// TIA Portal V19 export
FUNCTION_BLOCK "MwFakCalc_FB"   // FB145, LAD
TITLE = COIL CAR
// stored: MemoryReserve 100, SetENOAutomatically false
   VAR_INPUT
      AreaInterface : "AreaInterface";
      ZSI : "udt_ZoneSafetyInterface";
      DSI : Struct
         PushAx : "udt_DeviceSafetyInterface";
         Gripper : "udt_DeviceSafetyInterface";
      END_STRUCT;
      Drive : Struct
         PushAx : "TAx_DriveInterface";
      END_STRUCT;
      HWID : Struct
         PushAx_TEL1 : HW_SUBMODULE;
      END_STRUCT;
      DataIn : Struct
         MaterialPresenceEntry : Bool;
         MaterialPresenceExit : Bool;
         MaterialJam : Bool;
         PushAx_Ls_HomeFwd : Bool;
         PushAx_Ls_RestBwd : Bool;
         PushAx_Ls_LowSpeedHome : Bool;
         PushAx_Ls_LowSpeedRest : Bool;
         PushAx_Ls_Touch : Bool;
         Gripper_Ls_ForceOpen : Bool;   // TRUE = Movable supprts must be closed
         PushAx : "SpeedMachine_DataIn";
         Gripper : "ValveMachine_DataIn";
      END_STRUCT;
      CIn : Struct
         Manager : Struct
            EnableStopDoorOpeningReq : Bool;
            EnableStopInPhase : Bool;
            EnableStopProgrammed : Bool;
         END_STRUCT;
         Rollformer_Standstill : Bool;
         Rollformer_CheckNextFwd : Bool;
         Rollformer_CheckNextBwd : Bool;
         MW_ActualFAK : LReal;
         SemiAut_And_ButtonPressed : Bool;
         PostServo_MeasuredValueG : LReal;
         PostServo_MeasuredValueW : LReal;
         PostServo_MeasuredID : UInt;
      END_STRUCT;
      Config : Struct
         PushAx : "SpeedMachine_Config";
         Gripper : "ValveMachine_Config";
         MaterialPresenceDly : Time;
         MaterialAbsenceDly : Time;
         PushAx_FwdTimeout { ExternalAccessible := 'False'; ExternalVisible := 'False'; ExternalWritable := 'False'} : Time;
         PushAx_BwdTimeout { ExternalAccessible := 'False'; ExternalVisible := 'False'; ExternalWritable := 'False'} : Time;
         Default_FAK : LReal;
      END_STRUCT;
   END_VAR
   VAR_OUTPUT
      MachineInterface : "MachineInterface";
      DataOut : Struct
         PushAx : "SpeedMachine_DataOut";
         Gripper : "ValveMachine_DataOut";
         MeasInput_ExeReg : Bool;
      END_STRUCT;
      COut : Struct
         PushAx : "SpeedMachine_COut";
         Gripper : "ValveMachine_COut";
         StopMaterialFeeding : Bool;
         MW_FAK_ChangeIsRequest : Bool;
      END_STRUCT;
   END_VAR
   VAR_IN_OUT
      PersistentValues : "udt_MwFacCalc_Pers";
      TO_Gripper_Encoder : TO_ExternalEncoder;
      TO_Gripper_MeasInput : TO_MeasuringInput;
      TO_Wheel_MeasInput : TO_MeasuringInput;
   END_VAR
   VAR
      Sts : Struct
         PushAx : Struct
            LowSpeedRest : Bool;
            LowSpeedHome : Bool;
         END_STRUCT;
         Gripper : Struct
            OffsetPos : LReal;
            PosRel : LReal;
         END_STRUCT;
         AlarmPresence : Bool;
         Status : Int;
         MW_FAK_ChangeIsRequest : Bool;
         AverageFAKIsValid : Bool;
         WheelMeasInp_SaveIdLastPosEdge : UInt;
         GripperMeasInp_SaveIdLastPosEdge : UInt;
         GripperMeasInp_LastID : UInt;
         WheelMeasInp_LastID : UInt;
         PostServo_LastID : UInt;
      END_STRUCT;
      Ctrl : Struct
         StopInPhase : Bool;
         StopProgrammed : Bool;
         MeasuringStart : Bool;
         MeasInp_Enable : Bool;
         Meas1_Exe : Bool;
         Meas2_Exe : Bool;
         Gripper_RollformerForceOpen : Bool;
         Gripper_AutOpen : Bool;
         Gripper_AutClose : Bool;
         PushAx_AutFwd : Bool;
         PushAx_AutBwd : Bool;
         Rollformer_FwdEnable : Bool;
         Rollformer_BkwWnable : Bool;
         Rollformer_FastStop : Bool;
      END_STRUCT;
      Alarm : Struct
         PushAx_UnvalidStateLsZeroRest : Bool;
         PushAx_UnvalidStateLsLow : Bool;
         PushAx_LowSpeedHome_NotEngaged : Bool;
         PushAx_LowSpeedRest_NotEngaged : Bool;
         PushAx_TimeoutFwd : Bool;
         PushAx_TimeoutBwd : Bool;
         MaterialNoPresence : Bool;
         MaterialJamEntry : Bool;
         Meas1RegNotGet : Bool;
         Meas2RegNotGet : Bool;
         Gripper_MaxPosExceed : Bool;
         PushAx : "SpeedMachine_Alr";
         Gripper : "ValveAlr";
         Gripper_Encoder : "TExtEncoder_Alarms";
         Gripper_MeasInput : "TMeasuring_Alarms";
         Wheel_MeasInput : "TMeasuring_Alarms";
      END_STRUCT;
      Warning : Struct
         PushAx : "SpeedMachine_Wng";
         Gripper : "ValveMachine_Wng";
         MaterialNoPrresence : Bool;
      END_STRUCT;
      Diag : Struct
         Gripper_Encoder : "TO_Diagnostic";
         Gripper_MeasInput : "TO_Diagnostic";
         Wheel_MeasInput : "TO_Diagnostic";
      END_STRUCT;
      PushAx : "SpeedMachine_FB";
      Gripper : "ValveMachine_FB";
      Gripper_MeasInp { S7_SetPoint := 'True'} : "MeasuringInput";
      Wheel_MeasInp { S7_SetPoint := 'True'} : "MeasuringInput";
      MeasRegIEmpty { S7_SetPoint := 'True'} : "udt_MwFacCalc_RegItem";
      tonMaterialPresence : TON_TIME;
      tonMaterialAbsence : TON_TIME;
      tonPushAxFwd { S7_SetPoint := 'True'} : TON_TIME;
      tonPushAxBwd { S7_SetPoint := 'True'} : TON_TIME;
      tonRollformer_BwdCheckNext { S7_SetPoint := 'True'} : TON_TIME;
   END_VAR
   VAR_TEMP
      i : Int;
      Delta_W : LReal;
      Delta_G : LReal;
      FAK_Acc : LReal;
      Tol : LReal;
      LongerPartLength_ActualFAK : LReal;
      LongerPartLength_NewFAK : LReal;
   END_VAR
BEGIN

REGION Network 1 (SCL): Reset alarms command

   IF #AreaInterface.RstAlarms THEN
       // Alarms
       #Alarm.PushAx_UnvalidStateLsZeroRest := FALSE;
       #Alarm.PushAx_UnvalidStateLsLow := FALSE;
       #Alarm.PushAx_LowSpeedHome_NotEngaged := FALSE;
       #Alarm.PushAx_LowSpeedRest_NotEngaged := FALSE;
       #Alarm.PushAx_TimeoutFwd := FALSE;
       #Alarm.PushAx_TimeoutBwd := FALSE;
       #Alarm.MaterialNoPresence := FALSE;
       #Alarm.MaterialJamEntry := FALSE;
       #Alarm.Meas1RegNotGet := FALSE;
       #Alarm.Meas2RegNotGet := FALSE;
       #Alarm.Gripper_MaxPosExceed := FALSE;

   END_IF;
END_REGION

REGION Network 3: Material Presence
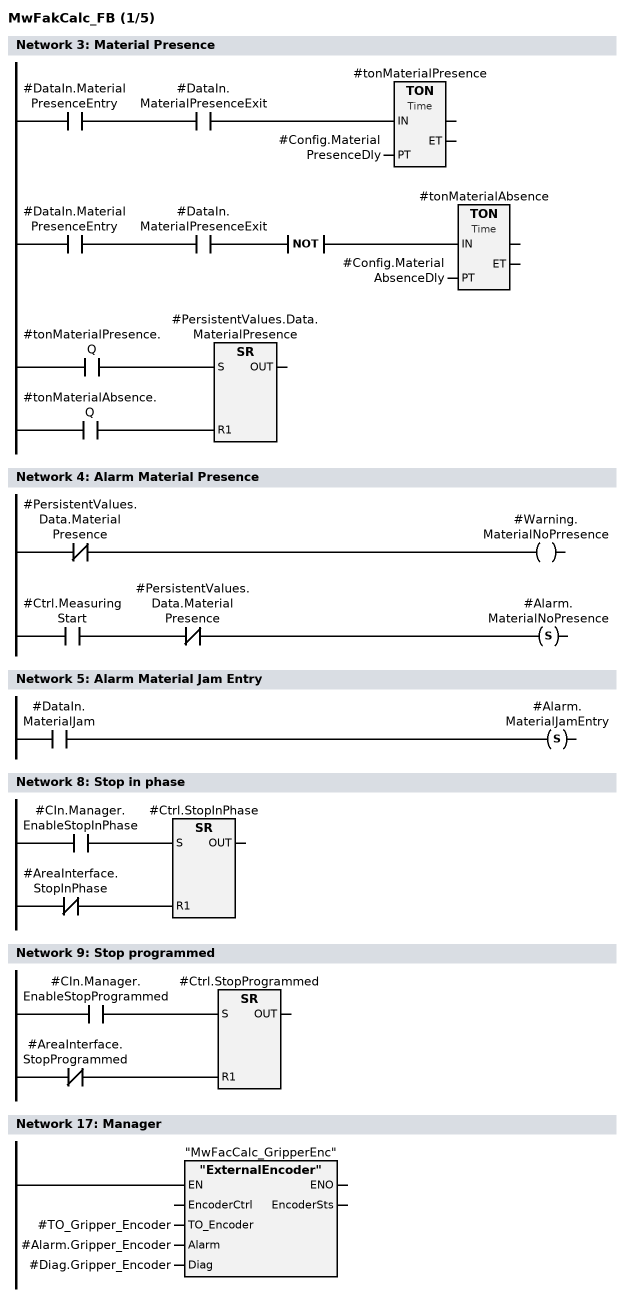
   RUNG wire#powerrail
      Contact( #DataIn.MaterialPresenceEntry )
      Contact( #DataIn.MaterialPresenceExit )
      { S7_Templates := "time_type := Time" } #tonMaterialPresence.TON(pt := #Config.MaterialPresenceDly, et =>)
   END_RUNG
   RUNG wire#powerrail
      Contact( #DataIn.MaterialPresenceEntry )
      Contact( #DataIn.MaterialPresenceExit )
      Not()
      { S7_Templates := "time_type := Time" } #tonMaterialAbsence.TON(pt := #Config.MaterialAbsenceDly, et =>)
   END_RUNG
   RUNG wire#powerrail
      Contact( #tonMaterialPresence.Q )
      S_SR(operand := #PersistentValues.Data.MaterialPresence, r1 := wire#w1)
   END_RUNG
   RUNG wire#powerrail
      Contact( #tonMaterialAbsence.Q )
   END_RUNG wire#w1
   // the same network as SCL:
   #tonMaterialPresence(IN := #DataIn.MaterialPresenceEntry AND #DataIn.MaterialPresenceExit,   // TON
                        PT := #Config.MaterialPresenceDly);
   #tonMaterialAbsence(IN := NOT (#DataIn.MaterialPresenceEntry AND #DataIn.MaterialPresenceExit),   // TON
                       PT := #Config.MaterialAbsenceDly);
   IF #tonMaterialPresence.Q THEN
       #PersistentValues.Data.MaterialPresence := TRUE;   // SR flip-flop
   END_IF;
   IF #tonMaterialAbsence.Q THEN #PersistentValues.Data.MaterialPresence := FALSE; END_IF;
END_REGION

REGION Network 4: Alarm Material Presence
   RUNG wire#powerrail
      I_Contact( #PersistentValues.Data.MaterialPresence )
      Coil( #Warning.MaterialNoPrresence )
   END_RUNG
   RUNG wire#powerrail
      Contact( #Ctrl.MeasuringStart )
      I_Contact( #PersistentValues.Data.MaterialPresence )
      S_Coil( #Alarm.MaterialNoPresence )
   END_RUNG
   // the same network as SCL:
   #Warning.MaterialNoPrresence := NOT #PersistentValues.Data.MaterialPresence;
   IF #Ctrl.MeasuringStart AND NOT #PersistentValues.Data.MaterialPresence THEN
       #Alarm.MaterialNoPresence := TRUE;
   END_IF;
END_REGION

REGION Network 5: Alarm Material Jam Entry
   RUNG wire#powerrail
      Contact( #DataIn.MaterialJam )
      S_Coil( #Alarm.MaterialJamEntry )
   END_RUNG
   // the same network as SCL:
   IF #DataIn.MaterialJam THEN #Alarm.MaterialJamEntry := TRUE; END_IF;
END_REGION

REGION Network 7: <<<CYCLE >>>
END_REGION

REGION Network 8: Stop in phase
   RUNG wire#powerrail
      Contact( #CIn.Manager.EnableStopInPhase )
      S_SR(operand := #Ctrl.StopInPhase, r1 := wire#w1)
   END_RUNG
   RUNG wire#powerrail
      I_Contact( #AreaInterface.StopInPhase )
   END_RUNG wire#w1
   // the same network as SCL:
   IF #CIn.Manager.EnableStopInPhase THEN
       #Ctrl.StopInPhase := TRUE;   // SR flip-flop
   END_IF;
   IF NOT #AreaInterface.StopInPhase THEN #Ctrl.StopInPhase := FALSE; END_IF;
END_REGION

REGION Network 9: Stop programmed
   RUNG wire#powerrail
      Contact( #CIn.Manager.EnableStopProgrammed )
      S_SR(operand := #Ctrl.StopProgrammed, r1 := wire#w1)
   END_RUNG
   RUNG wire#powerrail
      I_Contact( #AreaInterface.StopProgrammed )
   END_RUNG wire#w1
   // the same network as SCL:
   IF #CIn.Manager.EnableStopProgrammed THEN
       #Ctrl.StopProgrammed := TRUE;   // SR flip-flop
   END_IF;
   IF NOT #AreaInterface.StopProgrammed THEN #Ctrl.StopProgrammed := FALSE; END_IF;
END_REGION

REGION Network 10 (SCL): Start measure

   #tonRollformer_BwdCheckNext(IN := #CIn.Rollformer_CheckNextBwd,
                               PT := T#200ms);


   IF (#PersistentValues.Par.WorkMode = 0)
       OR
       #Sts.AlarmPresence
       OR
       #MachineInterface.AlarmsPresence
       OR
       #tonRollformer_BwdCheckNext.Q
       OR
       NOT #PersistentValues.Data.MaterialPresence
   THEN

       #Ctrl.MeasuringStart := FALSE;


   ELSIF #AreaInterface.Man AND #CIn.Rollformer_Standstill AND
       (#DataIn.Gripper.PB.Rest OR #DataIn.Gripper.PB.Work OR #DataIn.PushAx.PB.Bwd_Minus OR #DataIn.PushAx.PB.Fwd_Plus)
   THEN
       ;
       #Ctrl.MeasuringStart := FALSE;

   ELSIF #AreaInterface.Man AND #CIn.Rollformer_CheckNextFwd THEN
       #Ctrl.MeasuringStart := TRUE;

   ELSIF #AreaInterface.Aut THEN
       #Ctrl.MeasuringStart := TRUE;
   END_IF;


   IF #MachineInterface.AlarmsPresence OR (NOT #Ctrl.MeasuringStart AND #Sts.Status >= 30 AND #Sts.Status <= 90) THEN
       #Sts.Status := 90;
   END_IF;
END_REGION

REGION Network 11 (SCL): Sequence

   CASE #Sts.Status OF

           //INIT
       0:
           FOR #i := 1 TO "MWFAKCALC_REG_MAXITEM" DO
               #PersistentValues.Data.Reg[#i] := #MeasRegIEmpty;
           END_FOR;
           #PersistentValues.Data.RegItemsValid := 0;
           #Sts.Status += 1;

       1 : //IDLE 
           #Ctrl.Gripper_AutOpen := FALSE;
           #Ctrl.Gripper_AutClose := FALSE;
           #Ctrl.PushAx_AutFwd := FALSE;
           #Ctrl.PushAx_AutBwd := FALSE;
           #Ctrl.MeasInp_Enable := FALSE;
           #Ctrl.Meas1_Exe := FALSE;
           #Ctrl.Meas2_Exe := FALSE;

           IF #Ctrl.MeasuringStart THEN
               #Sts.Status := 30;

           ELSIF ((#PersistentValues.Par.WorkMode = 0) OR NOT #PersistentValues.Data.MaterialPresence) AND
               #PersistentValues.Data.Reg[1].ID <> 0
           THEN
               #Sts.Status := 0;
           END_IF;

       30: // Enable measuring input
           #Ctrl.MeasInp_Enable := TRUE;

           #Ctrl.Gripper_AutOpen := TRUE;
           #Ctrl.Gripper_AutClose := FALSE;

           IF #Gripper.COut.Rest AND
               #Gripper_MeasInp.MeasuringSts.InOperation AND
               #Wheel_MeasInp.MeasuringSts.InOperation
           THEN
               #Sts.Status += 1;
           END_IF;


       31://Pusher ax Fwd

           #Ctrl.PushAx_AutBwd := FALSE;

           IF NOT #DataIn.PushAx_Ls_HomeFwd THEN
               #Ctrl.PushAx_AutFwd := TRUE;
           ELSE
               #Ctrl.PushAx_AutFwd := FALSE;
               #Sts.Status := #Sts.Status + 1;
           END_IF;

       32: //Pusher ax Bwd

           #Ctrl.PushAx_AutFwd := FALSE;

           IF NOT #DataIn.PushAx_Ls_RestBwd THEN
               #Ctrl.PushAx_AutBwd := TRUE;
           ELSE
               #Ctrl.PushAx_AutBwd := FALSE;
               #Sts.Status += 1;
           END_IF;

       33: // Start measring cycle
           #Ctrl.Meas1_Exe := FALSE;
           #Ctrl.Meas2_Exe := FALSE;

           #Ctrl.Gripper_AutOpen := TRUE;
           #Ctrl.Gripper_AutClose := FALSE;

           IF #Gripper.COut.Rest AND
               #DataIn.PushAx_Ls_RestBwd
           THEN
               // Fine ciclo con misuratore in "ordine"    
               IF NOT #Ctrl.MeasuringStart THEN
                   #Sts.Status := 1;

                   // Avvio ciclo di misurazione   
               ELSE
                   #Ctrl.Gripper_AutClose := TRUE;
                   #Ctrl.Gripper_AutOpen := FALSE;
                   #Sts.Status += 1;
               END_IF;
           END_IF;

       34: // Command Meas 1

           IF #Gripper.COut.Work AND #Sts.Gripper.PosRel > #PersistentValues.Par.Gripper_Meas1_PosStart THEN

               #Sts.GripperMeasInp_LastID := #PersistentValues.Data.GripperMeasID;
               #Sts.WheelMeasInp_LastID := #PersistentValues.Data.WheelMeasID;
               #Sts.PostServo_LastID := #CIn.PostServo_MeasuredID;

               #Ctrl.Meas1_Exe := TRUE;
               #Sts.Status += 1;
           END_IF;

       35: // Detect Meas 1

           IF #Sts.GripperMeasInp_LastID <> #PersistentValues.Data.GripperMeasID AND
               #Sts.WheelMeasInp_LastID <> #PersistentValues.Data.WheelMeasID AND
               #CIn.PostServo_MeasuredID <> #Sts.PostServo_LastID
           THEN
               #Ctrl.Meas1_Exe := FALSE;

               IF #PersistentValues.Data.RegID <= 0 THEN
                   #PersistentValues.Data.RegID := 1;
               END_IF;

               // Shift in basso per liberare prima posizione
               #i := "MWFAKCALC_REG_MAXITEM" - 1;

               WHILE #i >= 1 DO
                   #PersistentValues.Data.Reg[#i + 1] := #PersistentValues.Data.Reg[#i];
                   #i -= 1;
               END_WHILE;

               // Cancellazione vecchi valori
               #PersistentValues.Data.Reg[1] := #MeasRegIEmpty;

               // Iserimento valori inizio misurazione
               #PersistentValues.Data.Reg[1].ID := #PersistentValues.Data.RegID;
               #PersistentValues.Data.Reg[1].TP_W_Meas1Reg.ID := #PersistentValues.Data.WheelMeasID;
               #PersistentValues.Data.Reg[1].TP_W_Meas1Reg.Position := #Wheel_MeasInp.MeasuringSts.MeasuringValue1;
               #PersistentValues.Data.Reg[1].TP_G_Meas1Reg.ID := #PersistentValues.Data.GripperMeasID;
               #PersistentValues.Data.Reg[1].TP_G_Meas1Reg.Position := #Gripper_MeasInp.MeasuringSts.MeasuringValue1;

               //Measured Post servo
               #PersistentValues.Data.Reg[1].PS_W_Meas1Reg.ID := #CIn.PostServo_MeasuredID;
               #PersistentValues.Data.Reg[1].PS_W_Meas1Reg.Position := #CIn.PostServo_MeasuredValueW;
               #PersistentValues.Data.Reg[1].PS_G_Meas1Reg.ID := #CIn.PostServo_MeasuredID;
               #PersistentValues.Data.Reg[1].PS_G_Meas1Reg.Position := #CIn.PostServo_MeasuredValueG;

               #PersistentValues.Data.RegID += 1;

               #Sts.WheelMeasInp_SaveIdLastPosEdge := #PersistentValues.Data.Reg[1].TP_W_Meas1Reg.ID;
               #Sts.GripperMeasInp_SaveIdLastPosEdge := #PersistentValues.Data.Reg[1].TP_G_Meas1Reg.ID;
               #Sts.Status += 1;

           ELSIF #Sts.Gripper.PosRel > #PersistentValues.Par.Gripper_Meas1_DonePosLim THEN
               #Alarm.Meas1RegNotGet := TRUE;
               "A02_DEBUG".MwFakCalc.GripperPosRel := #Sts.Gripper.PosRel;
               #Sts.Status := 90;

           END_IF;

       36: //Command Meas 2
           IF #Gripper.COut.Work AND #Sts.Gripper.PosRel > #PersistentValues.Par.Gripper_Meas2_PosStart THEN
               #Sts.GripperMeasInp_LastID := #PersistentValues.Data.GripperMeasID;
               #Sts.WheelMeasInp_LastID := #PersistentValues.Data.WheelMeasID;
               #Sts.PostServo_LastID := #CIn.PostServo_MeasuredID;

               #Ctrl.Meas2_Exe := TRUE;
               #Sts.Status += 1;
           END_IF;


       37: //Detect Meas 2
           IF  #Sts.GripperMeasInp_LastID <> #PersistentValues.Data.GripperMeasID AND
               #Sts.WheelMeasInp_LastID <> #PersistentValues.Data.WheelMeasID AND
               #CIn.PostServo_MeasuredID <> #Sts.PostServo_LastID
           THEN

               // Inserimento valori fine misurazione  
               #PersistentValues.Data.Reg[1].TP_W_Meas2Reg.ID := #PersistentValues.Data.WheelMeasID;
               #PersistentValues.Data.Reg[1].TP_W_Meas2Reg.Position := #Wheel_MeasInp.MeasuringSts.MeasuringValue1;
               #PersistentValues.Data.Reg[1].TP_G_Meas2Reg.ID := #PersistentValues.Data.GripperMeasID;
               #PersistentValues.Data.Reg[1].TP_G_Meas2Reg.Position := #Gripper_MeasInp.MeasuringSts.MeasuringValue1;

               //Measured Post servo
               #PersistentValues.Data.Reg[1].PS_W_Meas2Reg.ID := #CIn.PostServo_MeasuredID;
               #PersistentValues.Data.Reg[1].PS_W_Meas2Reg.Position := #CIn.PostServo_MeasuredValueW;
               #PersistentValues.Data.Reg[1].PS_G_Meas2Reg.ID := #CIn.PostServo_MeasuredID;
               #PersistentValues.Data.Reg[1].PS_G_Meas2Reg.Position := #CIn.PostServo_MeasuredValueG;

               #Sts.Status += 1;

           ELSIF #Sts.Gripper.PosRel > #PersistentValues.Par.Gripper_Meas2_DonePosLim THEN
               #Alarm.Meas2RegNotGet := TRUE;
               #Sts.Status := 90;

           END_IF;

       38: //Caluclate Average FAK

           #Delta_W := "M_PosAMinusPosB"(PosA := #PersistentValues.Data.Reg[1].TP_W_Meas2Reg.Position, PosB := #PersistentValues.Data.Reg[1].TP_W_Meas1Reg.Position, MODULE := "MATERIAL_COUNTERS_MODULE");
           #Delta_G := #PersistentValues.Data.Reg[1].TP_G_Meas2Reg.Position - #PersistentValues.Data.Reg[1].TP_G_Meas1Reg.Position;
           #PersistentValues.Data.Reg[1].TP_DeltaW := #Delta_W;
           #PersistentValues.Data.Reg[1].TP_DeltaG := #Delta_G;

           IF #Delta_W <> 0 AND #Delta_G <> 0 THEN
               #PersistentValues.Data.Reg[1].FAK := #Delta_G / #Delta_W;
           ELSE
               #PersistentValues.Data.Reg[1].FAK := 0.0;
           END_IF;


           //Post servo average FAK
           #Delta_W := "M_PosAMinusPosB"(PosA := #PersistentValues.Data.Reg[1].PS_W_Meas2Reg.Position, PosB := #PersistentValues.Data.Reg[1].PS_W_Meas1Reg.Position, MODULE := "MATERIAL_COUNTERS_MODULE");
           #Delta_G := #PersistentValues.Data.Reg[1].PS_G_Meas2Reg.Position - #PersistentValues.Data.Reg[1].PS_G_Meas1Reg.Position;
           #PersistentValues.Data.Reg[1].PS_DeltaW := #Delta_W;
           #PersistentValues.Data.Reg[1].PS_DeltaG := #Delta_G;

           IF #Delta_W <> 0 AND #Delta_G <> 0 THEN
               #PersistentValues.Data.Reg[1].FAK_PS := #Delta_G / #Delta_W;
           ELSE
               #PersistentValues.Data.Reg[1].FAK_PS := 0.0;
           END_IF;


           #PersistentValues.Data.RegItemsValid := 0;
           #FAK_Acc := 0;


           FOR #i := 1 TO "MWFAKCALC_REG_MAXITEM" DO
               IF #PersistentValues.Data.Reg[#i].FAK > "FAK_MIN_VALUE" AND #PersistentValues.Data.Reg[#i].FAK < "FAK_MAX_VALUE"
               THEN
                   #PersistentValues.Data.RegItemsValid := #PersistentValues.Data.RegItemsValid + 1;
                   #FAK_Acc := #FAK_Acc + #PersistentValues.Data.Reg[#i].FAK;
               END_IF;

               IF #PersistentValues.Data.RegItemsValid > 0
               THEN
                   #PersistentValues.Data.AverageFAK := #FAK_Acc / #PersistentValues.Data.RegItemsValid;
               ELSE
                   #PersistentValues.Data.AverageFAK := #Config.Default_FAK;
               END_IF;
           END_FOR;

           #Ctrl.Gripper_AutOpen := TRUE;
           #Ctrl.Gripper_AutClose := FALSE;
           #Ctrl.Meas2_Exe := FALSE;

           #Sts.Status := 30;


       90: // STOP

           #Ctrl.Gripper_AutOpen := NOT #Gripper.COut.Rest;
           #Ctrl.Gripper_AutClose := FALSE;
           #Ctrl.PushAx_AutBwd := FALSE;
           #Ctrl.PushAx_AutFwd := FALSE;

           IF NOT #MachineInterface.AlarmsPresence AND #Gripper.COut.Rest THEN
               #Sts.Status := 1;
           END_IF;
   END_CASE;
END_REGION

REGION Network 12 (SCL): Caluclate new FAK

   // Se il calcolo della media non è corretto è assegnato il valore di default !
   IF #PersistentValues.Data.RegItemsValid < 1 OR #PersistentValues.Data.AverageFAK <= "FAK_MIN_VALUE" OR #PersistentValues.Data.AverageFAK >= "FAK_MAX_VALUE"
   THEN
       #PersistentValues.Data.AverageFAK := #Config.Default_FAK;
   END_IF;


   #Sts.AverageFAKIsValid := #PersistentValues.Data.RegItemsValid >= 1 AND #PersistentValues.Data.AverageFAK > "FAK_MIN_VALUE" AND #PersistentValues.Data.AverageFAK < "FAK_MAX_VALUE";

   IF #Sts.AverageFAKIsValid THEN
       #LongerPartLength_NewFAK := "P_LEN_MAX" * #PersistentValues.Data.AverageFAK;

       IF #CIn.Rollformer_Standstill AND NOT #CIn.SemiAut_And_ButtonPressed
       THEN
           #Tol := 0.01;
       ELSE
           #Tol := 0.1;
       END_IF;

       // Il FAK deve essere cambiato sulla ruota di misura MLC per mantenere l'errore di misura inferiore a 0.1 mm
       #LongerPartLength_ActualFAK := "P_LEN_MAX" * #CIn.MW_ActualFAK;

       #Sts.MW_FAK_ChangeIsRequest := ABS(#LongerPartLength_NewFAK - #LongerPartLength_ActualFAK) > #Tol;
   ELSE
       #Sts.MW_FAK_ChangeIsRequest := FALSE;
   END_IF;
END_REGION

REGION Network 14: <<< GRIPPER ENCODER>>>
END_REGION

REGION Network 15 (SCL): Gripper relative position
   // Posizione pinza relativa..si azzera quando la pinza è sul fc di home
   IF #DataIn.PushAx_Ls_LowSpeedHome OR #DataIn.PushAx_Ls_HomeFwd
   THEN
       #Sts.Gripper.OffsetPos := #TO_Gripper_Encoder.ActualPosition;
   END_IF;

   #Sts.Gripper.PosRel := #TO_Gripper_Encoder.ActualPosition - #Sts.Gripper.OffsetPos;
END_REGION

REGION Network 16 (SCL): Control
   "MwFacCalc_GripperEnc".EncoderCtrl.Rst := #AreaInterface.RstAlarms;
END_REGION

REGION Network 17: Manager
   RUNG wire#powerrail
      "MwFacCalc_GripperEnc"(EncoderCtrl :=, TO_Encoder := #TO_Gripper_Encoder, Alarm := #Alarm.Gripper_Encoder, Diag := #Diag.Gripper_Encoder, EncoderSts =>)
   END_RUNG
   // the same network as SCL:
   "MwFacCalc_GripperEnc"(TO_Encoder := #TO_Gripper_Encoder,   // "ExternalEncoder"
                          Alarm := #Alarm.Gripper_Encoder,
                          Diag := #Diag.Gripper_Encoder);
END_REGION

REGION Network 18: >
END_REGION

REGION Network 19: <<< GRIPPER MEAS INPUT >>>
END_REGION

REGION Network 20 (SCL): Control
   #Gripper_MeasInp.MeasuringCtrl.Rst := #AreaInterface.RstAlarms;
   #Gripper_MeasInp.MeasuringCtrl.MeasureEnable := #Ctrl.MeasInp_Enable;
   #Gripper_MeasInp.MeasuringCtrl.Mode := 0;
END_REGION

REGION Network 21: Manager
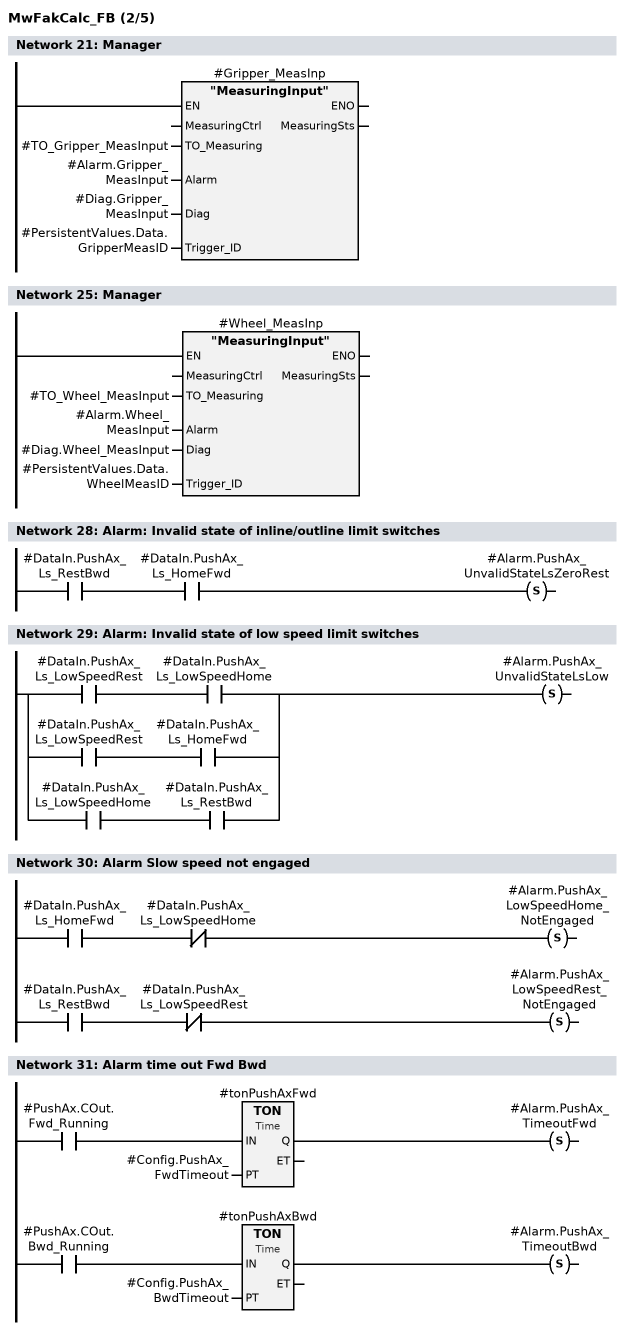
   RUNG wire#powerrail
      #Gripper_MeasInp(MeasuringCtrl :=, TO_Measuring := #TO_Gripper_MeasInput, Alarm := #Alarm.Gripper_MeasInput, Diag := #Diag.Gripper_MeasInput, Trigger_ID := #PersistentValues.Data.GripperMeasID, MeasuringSts =>)
   END_RUNG
   // the same network as SCL:
   #Gripper_MeasInp(TO_Measuring := #TO_Gripper_MeasInput,   // "MeasuringInput"
                    Alarm := #Alarm.Gripper_MeasInput,
                    Diag := #Diag.Gripper_MeasInput,
                    Trigger_ID := #PersistentValues.Data.GripperMeasID);
END_REGION

REGION Network 22: >
END_REGION

REGION Network 23: <<< WHEEL MEAS INPUT >>>
END_REGION

REGION Network 24 (SCL): Control
   #Wheel_MeasInp.MeasuringCtrl.Rst := #AreaInterface.RstAlarms;
   #Wheel_MeasInp.MeasuringCtrl.MeasureEnable := #Ctrl.MeasInp_Enable;
   #Wheel_MeasInp.MeasuringCtrl.Mode := 0;
END_REGION

REGION Network 25: Manager
   RUNG wire#powerrail
      #Wheel_MeasInp(MeasuringCtrl :=, TO_Measuring := #TO_Wheel_MeasInput, Alarm := #Alarm.Wheel_MeasInput, Diag := #Diag.Wheel_MeasInput, Trigger_ID := #PersistentValues.Data.WheelMeasID, MeasuringSts =>)
   END_RUNG
   // the same network as SCL:
   #Wheel_MeasInp(TO_Measuring := #TO_Wheel_MeasInput,   // "MeasuringInput"
                  Alarm := #Alarm.Wheel_MeasInput,
                  Diag := #Diag.Wheel_MeasInput,
                  Trigger_ID := #PersistentValues.Data.WheelMeasID);
END_REGION

REGION Network 26: >
END_REGION

REGION Network 27: <<< PUSH AX >>>
END_REGION

REGION Network 28: Alarm: Invalid state of inline/outline limit switches
   RUNG wire#powerrail
      Contact( #DataIn.PushAx_Ls_RestBwd )
      Contact( #DataIn.PushAx_Ls_HomeFwd )
      S_Coil( #Alarm.PushAx_UnvalidStateLsZeroRest )
   END_RUNG
   // the same network as SCL:
   IF #DataIn.PushAx_Ls_RestBwd AND #DataIn.PushAx_Ls_HomeFwd THEN
       #Alarm.PushAx_UnvalidStateLsZeroRest := TRUE;
   END_IF;
END_REGION

REGION Network 29: Alarm: Invalid state of low speed limit switches
   RUNG wire#powerrail
      Contact( #DataIn.PushAx_Ls_LowSpeedRest )
      Contact( #DataIn.PushAx_Ls_LowSpeedHome )
      wire#w1
      S_Coil( #Alarm.PushAx_UnvalidStateLsLow )
   END_RUNG
   RUNG wire#powerrail
      Contact( #DataIn.PushAx_Ls_LowSpeedRest )
      Contact( #DataIn.PushAx_Ls_HomeFwd )
   END_RUNG wire#w1
   RUNG wire#powerrail
      Contact( #DataIn.PushAx_Ls_LowSpeedHome )
      Contact( #DataIn.PushAx_Ls_RestBwd )
   END_RUNG wire#w1
   // the same network as SCL:
   IF (#DataIn.PushAx_Ls_LowSpeedRest AND #DataIn.PushAx_Ls_LowSpeedHome) OR (#DataIn.PushAx_Ls_LowSpeedRest AND #DataIn.PushAx_Ls_HomeFwd) OR (#DataIn.PushAx_Ls_LowSpeedHome AND #DataIn.PushAx_Ls_RestBwd) THEN
       #Alarm.PushAx_UnvalidStateLsLow := TRUE;
   END_IF;
END_REGION

REGION Network 30: Alarm Slow speed not engaged
   RUNG wire#powerrail
      Contact( #DataIn.PushAx_Ls_HomeFwd )
      I_Contact( #DataIn.PushAx_Ls_LowSpeedHome )
      S_Coil( #Alarm.PushAx_LowSpeedHome_NotEngaged )
   END_RUNG
   RUNG wire#powerrail
      Contact( #DataIn.PushAx_Ls_RestBwd )
      I_Contact( #DataIn.PushAx_Ls_LowSpeedRest )
      S_Coil( #Alarm.PushAx_LowSpeedRest_NotEngaged )
   END_RUNG
   // the same network as SCL:
   IF #DataIn.PushAx_Ls_HomeFwd AND NOT #DataIn.PushAx_Ls_LowSpeedHome THEN
       #Alarm.PushAx_LowSpeedHome_NotEngaged := TRUE;
   END_IF;
   IF #DataIn.PushAx_Ls_RestBwd AND NOT #DataIn.PushAx_Ls_LowSpeedRest THEN
       #Alarm.PushAx_LowSpeedRest_NotEngaged := TRUE;
   END_IF;
END_REGION

REGION Network 31: Alarm time out Fwd Bwd
   RUNG wire#powerrail
      Contact( #PushAx.COut.Fwd_Running )
      { S7_Templates := "time_type := Time" } #tonPushAxFwd.TON(pt := #Config.PushAx_FwdTimeout, et =>)
      S_Coil( #Alarm.PushAx_TimeoutFwd )
   END_RUNG
   RUNG wire#powerrail
      Contact( #PushAx.COut.Bwd_Running )
      { S7_Templates := "time_type := Time" } #tonPushAxBwd.TON(pt := #Config.PushAx_BwdTimeout, et =>)
      S_Coil( #Alarm.PushAx_TimeoutBwd )
   END_RUNG
   // the same network as SCL:
   #tonPushAxFwd(IN := #PushAx.COut.Fwd_Running, PT := #Config.PushAx_FwdTimeout);   // TON
   IF #tonPushAxFwd.Q THEN #Alarm.PushAx_TimeoutFwd := TRUE; END_IF;
   #tonPushAxBwd(IN := #PushAx.COut.Bwd_Running, PT := #Config.PushAx_BwdTimeout);   // TON
   IF #tonPushAxBwd.Q THEN #Alarm.PushAx_TimeoutBwd := TRUE; END_IF;
END_REGION

REGION Network 32: Move is in low speed
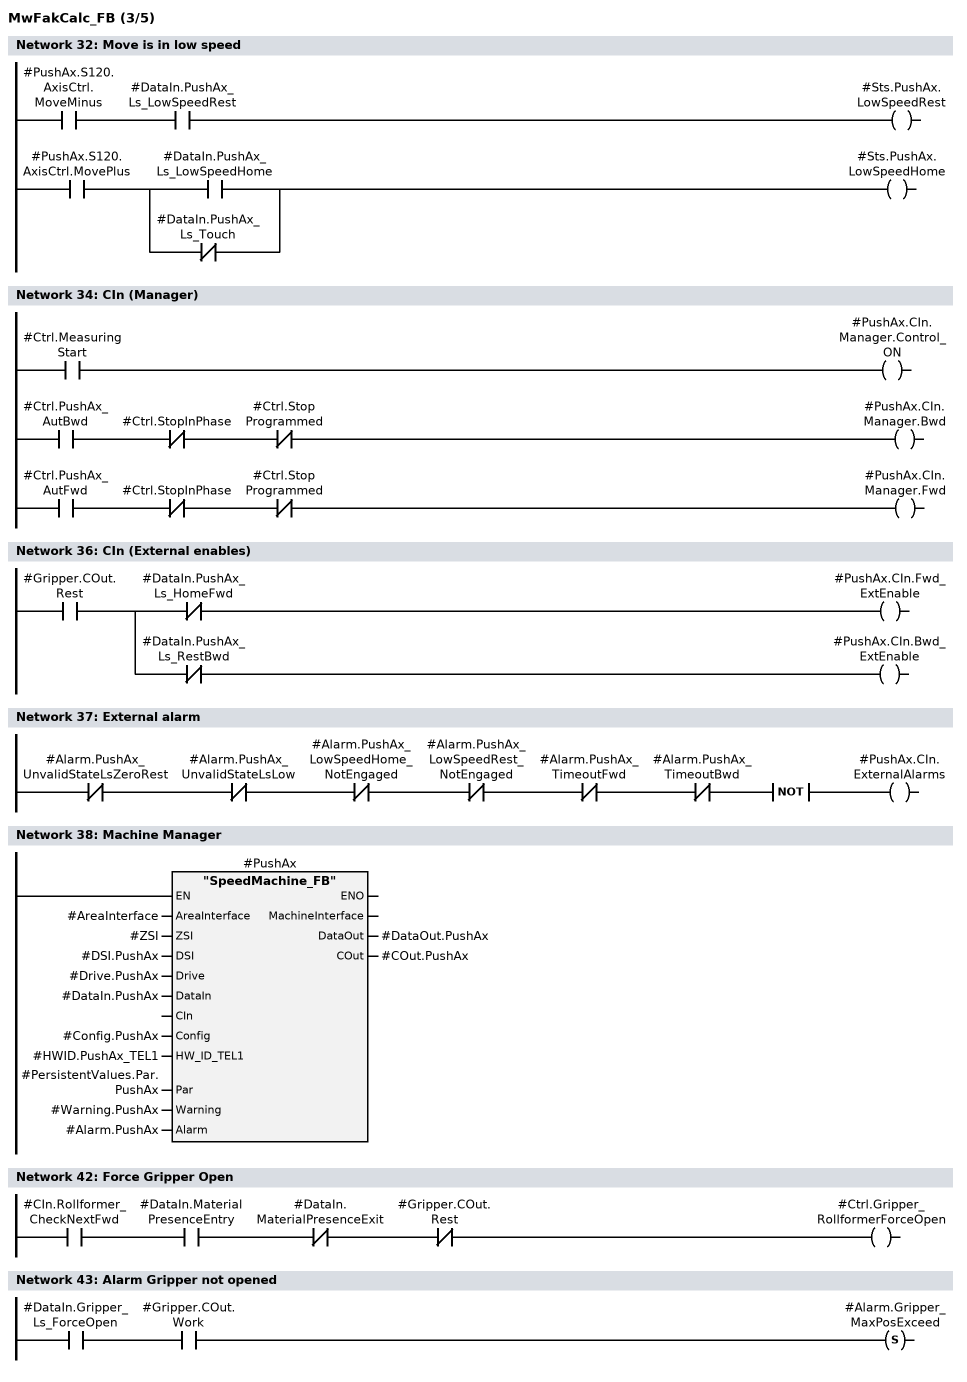
   RUNG wire#powerrail
      Contact( #PushAx.S120.AxisCtrl.MoveMinus )
      Contact( #DataIn.PushAx_Ls_LowSpeedRest )
      Coil( #Sts.PushAx.LowSpeedRest )
   END_RUNG
   RUNG wire#powerrail
      Contact( #PushAx.S120.AxisCtrl.MovePlus )
      wire#w1
      Contact( #DataIn.PushAx_Ls_LowSpeedHome )
      wire#w2
      Coil( #Sts.PushAx.LowSpeedHome )
   END_RUNG
   RUNG wire#w1
      I_Contact( #DataIn.PushAx_Ls_Touch )
   END_RUNG wire#w2
   // the same network as SCL:
   #Sts.PushAx.LowSpeedRest := #PushAx.S120.AxisCtrl.MoveMinus AND #DataIn.PushAx_Ls_LowSpeedRest;
   #Sts.PushAx.LowSpeedHome := #PushAx.S120.AxisCtrl.MovePlus AND (#DataIn.PushAx_Ls_LowSpeedHome OR NOT #DataIn.PushAx_Ls_Touch);
END_REGION

REGION Network 33 (SCL): Cin (Manager stop)
   #PushAx.CIn.Manager.EnableStopDoorOpeningReq := #CIn.Manager.EnableStopDoorOpeningReq;
   #PushAx.CIn.Manager.EnableStopInPhase := #Ctrl.StopInPhase;
   #PushAx.CIn.Manager.EnableStopProgrammed := #Ctrl.StopProgrammed;
END_REGION

REGION Network 34: CIn (Manager)
   RUNG wire#powerrail
      Contact( #Ctrl.MeasuringStart )
      Coil( #PushAx.CIn.Manager.Control_ON )
   END_RUNG
   RUNG wire#powerrail
      Contact( #Ctrl.PushAx_AutBwd )
      I_Contact( #Ctrl.StopInPhase )
      I_Contact( #Ctrl.StopProgrammed )
      Coil( #PushAx.CIn.Manager.Bwd )
   END_RUNG
   RUNG wire#powerrail
      Contact( #Ctrl.PushAx_AutFwd )
      I_Contact( #Ctrl.StopInPhase )
      I_Contact( #Ctrl.StopProgrammed )
      Coil( #PushAx.CIn.Manager.Fwd )
   END_RUNG
   // the same network as SCL:
   #PushAx.CIn.Manager.Control_ON := #Ctrl.MeasuringStart;
   #PushAx.CIn.Manager.Bwd := #Ctrl.PushAx_AutBwd AND NOT #Ctrl.StopInPhase AND NOT #Ctrl.StopProgrammed;
   #PushAx.CIn.Manager.Fwd := #Ctrl.PushAx_AutFwd AND NOT #Ctrl.StopInPhase AND NOT #Ctrl.StopProgrammed;
END_REGION

REGION Network 35 (SCL): Cin Dynamic

   //Automatic 
   IF #Sts.PushAx.LowSpeedRest OR #Sts.PushAx.LowSpeedHome THEN
       #PushAx.CIn.Manager.Vel := #PersistentValues.Par.PushAx_Aut_VelLow;
   ELSE
       #PushAx.CIn.Manager.Vel := #PersistentValues.Par.PushAx_Aut_VelHigh;
   END_IF;
   #PushAx.CIn.Manager.Acc := #PersistentValues.Par.PushAx_Aut_Acc;
   #PushAx.CIn.Manager.Dec := #PersistentValues.Par.PushAx_Aut_Dec;


   //Manual
   #PushAx.CIn.EnableManChangeVel := NOT #Sts.PushAx.LowSpeedRest AND NOT #Sts.PushAx.LowSpeedHome;
   #PersistentValues.Par.PushAx.Man.DelayChangeVel := T#1mS;
END_REGION

REGION Network 36: CIn (External enables)
   RUNG wire#powerrail
      Contact( #Gripper.COut.Rest )
      wire#w1
      I_Contact( #DataIn.PushAx_Ls_HomeFwd )
      Coil( #PushAx.CIn.Fwd_ExtEnable )
   END_RUNG
   RUNG wire#w1
      I_Contact( #DataIn.PushAx_Ls_RestBwd )
      Coil( #PushAx.CIn.Bwd_ExtEnable )
   END_RUNG
   // the same network as SCL:
   #PushAx.CIn.Fwd_ExtEnable := #Gripper.COut.Rest AND NOT #DataIn.PushAx_Ls_HomeFwd;
   #PushAx.CIn.Bwd_ExtEnable := #Gripper.COut.Rest AND NOT #DataIn.PushAx_Ls_RestBwd;
END_REGION

REGION Network 37: External alarm
   RUNG wire#powerrail
      I_Contact( #Alarm.PushAx_UnvalidStateLsZeroRest )
      I_Contact( #Alarm.PushAx_UnvalidStateLsLow )
      I_Contact( #Alarm.PushAx_LowSpeedHome_NotEngaged )
      I_Contact( #Alarm.PushAx_LowSpeedRest_NotEngaged )
      I_Contact( #Alarm.PushAx_TimeoutFwd )
      I_Contact( #Alarm.PushAx_TimeoutBwd )
      Not()
      Coil( #PushAx.CIn.ExternalAlarms )
   END_RUNG
   // the same network as SCL:
   #PushAx.CIn.ExternalAlarms := NOT (NOT #Alarm.PushAx_UnvalidStateLsZeroRest AND NOT #Alarm.PushAx_UnvalidStateLsLow AND NOT #Alarm.PushAx_LowSpeedHome_NotEngaged AND NOT #Alarm.PushAx_LowSpeedRest_NotEngaged AND NOT #Alarm.PushAx_TimeoutFwd AND NOT #Alarm.PushAx_TimeoutBwd);
END_REGION

REGION Network 38: Machine Manager
   RUNG wire#powerrail
      #PushAx(AreaInterface := #AreaInterface, ZSI := #ZSI, DSI := #DSI.PushAx, Drive := #Drive.PushAx, DataIn := #DataIn.PushAx, CIn :=, Config := #Config.PushAx, HW_ID_TEL1 := #HWID.PushAx_TEL1, Par := #PersistentValues.Par.PushAx, Warning := #Warning.PushAx, Alarm := #Alarm.PushAx, MachineInterface =>, DataOut => #DataOut.PushAx, COut => #COut.PushAx)
   END_RUNG
   // the same network as SCL:
   #PushAx(AreaInterface := #AreaInterface,   // "SpeedMachine_FB"
           ZSI := #ZSI,
           DSI := #DSI.PushAx,
           Drive := #Drive.PushAx,
           DataIn := #DataIn.PushAx,
           Config := #Config.PushAx,
           HW_ID_TEL1 := #HWID.PushAx_TEL1,
           Par := #PersistentValues.Par.PushAx,
           Warning := #Warning.PushAx,
           Alarm := #Alarm.PushAx,
           DataOut => #DataOut.PushAx,
           COut => #COut.PushAx);
END_REGION

REGION Network 39: >
END_REGION

REGION Network 40: >
END_REGION

REGION Network 41: <<< GRIPPER >>>
END_REGION

REGION Network 42: Force Gripper Open
   RUNG wire#powerrail
      Contact( #CIn.Rollformer_CheckNextFwd )
      Contact( #DataIn.MaterialPresenceEntry )
      I_Contact( #DataIn.MaterialPresenceExit )
      I_Contact( #Gripper.COut.Rest )
      Coil( #Ctrl.Gripper_RollformerForceOpen )
   END_RUNG
   // the same network as SCL:
   #Ctrl.Gripper_RollformerForceOpen := #CIn.Rollformer_CheckNextFwd AND #DataIn.MaterialPresenceEntry AND NOT #DataIn.MaterialPresenceExit AND NOT #Gripper.COut.Rest;
END_REGION

REGION Network 43: Alarm Gripper not opened
   RUNG wire#powerrail
      Contact( #DataIn.Gripper_Ls_ForceOpen )
      Contact( #Gripper.COut.Work )
      S_Coil( #Alarm.Gripper_MaxPosExceed )
   END_RUNG
   // the same network as SCL:
   IF #DataIn.Gripper_Ls_ForceOpen AND #Gripper.COut.Work THEN #Alarm.Gripper_MaxPosExceed := TRUE; END_IF;
END_REGION

REGION Network 44 (SCL): Cin (Manager stop)
   #Gripper.Cin.Manager.EnableStopDoorOpeningReq := #CIn.Manager.EnableStopDoorOpeningReq;
   #Gripper.Cin.Manager.EnableStopInPhase := #Ctrl.StopInPhase;
   #Gripper.Cin.Manager.EnableStopProgrammed := #Ctrl.StopProgrammed;
END_REGION

REGION Network 45: CIn (external enables)
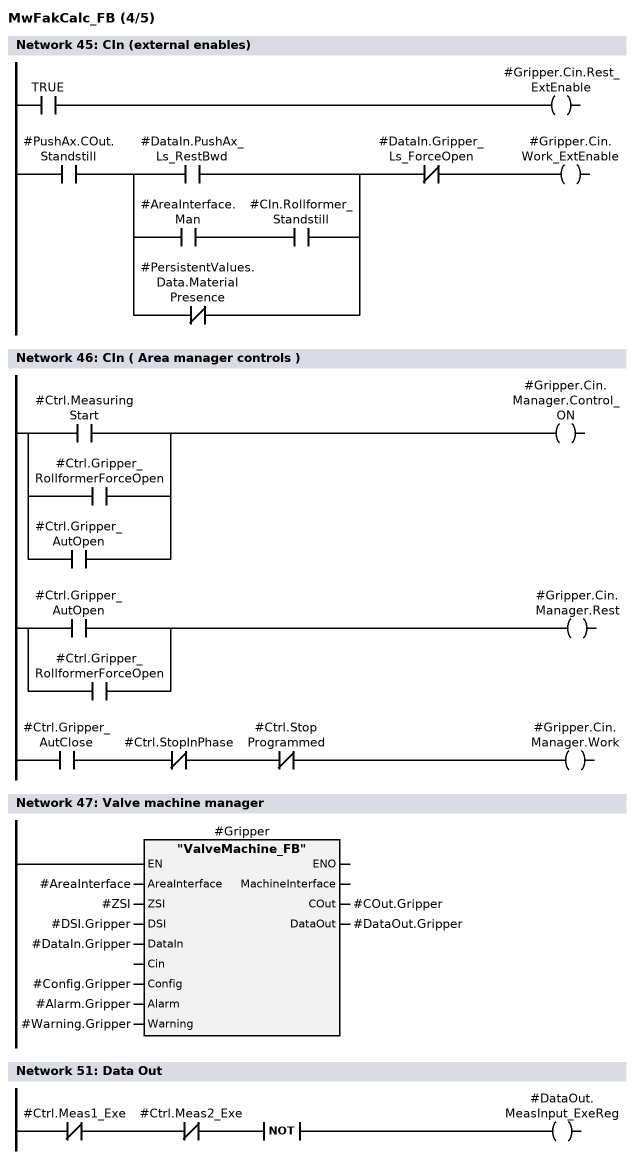
   RUNG wire#powerrail
      Contact( TRUE )
      Coil( #Gripper.Cin.Rest_ExtEnable )
   END_RUNG
   RUNG wire#powerrail
      Contact( #PushAx.COut.Standstill )
      wire#w1
      Contact( #DataIn.PushAx_Ls_RestBwd )
      wire#w2
      I_Contact( #DataIn.Gripper_Ls_ForceOpen )
      Coil( #Gripper.Cin.Work_ExtEnable )
   END_RUNG
   RUNG wire#w1
      Contact( #AreaInterface.Man )
      Contact( #CIn.Rollformer_Standstill )
   END_RUNG wire#w2
   RUNG wire#w1
      I_Contact( #PersistentValues.Data.MaterialPresence )
   END_RUNG wire#w2
   // the same network as SCL:
   #Gripper.Cin.Rest_ExtEnable := TRUE;
   #Gripper.Cin.Work_ExtEnable := #PushAx.COut.Standstill AND (#DataIn.PushAx_Ls_RestBwd OR (#AreaInterface.Man AND #CIn.Rollformer_Standstill) OR NOT #PersistentValues.Data.MaterialPresence) AND NOT #DataIn.Gripper_Ls_ForceOpen;
END_REGION

REGION Network 46: CIn ( Area manager controls )
   RUNG wire#powerrail
      Contact( #Ctrl.MeasuringStart )
      wire#w1
      Coil( #Gripper.Cin.Manager.Control_ON )
   END_RUNG
   RUNG wire#powerrail
      Contact( #Ctrl.Gripper_RollformerForceOpen )
   END_RUNG wire#w1
   RUNG wire#powerrail
      Contact( #Ctrl.Gripper_AutOpen )
   END_RUNG wire#w1
   RUNG wire#powerrail
      Contact( #Ctrl.Gripper_AutOpen )
      wire#w2
      Coil( #Gripper.Cin.Manager.Rest )
   END_RUNG
   RUNG wire#powerrail
      Contact( #Ctrl.Gripper_RollformerForceOpen )
   END_RUNG wire#w2
   RUNG wire#powerrail
      Contact( #Ctrl.Gripper_AutClose )
      I_Contact( #Ctrl.StopInPhase )
      I_Contact( #Ctrl.StopProgrammed )
      Coil( #Gripper.Cin.Manager.Work )
   END_RUNG
   // the same network as SCL:
   #Gripper.Cin.Manager.Control_ON := #Ctrl.MeasuringStart OR #Ctrl.Gripper_RollformerForceOpen OR #Ctrl.Gripper_AutOpen;
   #Gripper.Cin.Manager.Rest := #Ctrl.Gripper_AutOpen OR #Ctrl.Gripper_RollformerForceOpen;
   #Gripper.Cin.Manager.Work := #Ctrl.Gripper_AutClose AND NOT #Ctrl.StopInPhase AND NOT #Ctrl.StopProgrammed;
END_REGION

REGION Network 47: Valve machine manager
   RUNG wire#powerrail
      #Gripper(AreaInterface := #AreaInterface, ZSI := #ZSI, DSI := #DSI.Gripper, DataIn := #DataIn.Gripper, Cin :=, Config := #Config.Gripper, Alarm := #Alarm.Gripper, Warning := #Warning.Gripper, MachineInterface =>, COut => #COut.Gripper, DataOut => #DataOut.Gripper)
   END_RUNG
   // the same network as SCL:
   #Gripper(AreaInterface := #AreaInterface,   // "ValveMachine_FB"
            ZSI := #ZSI,
            DSI := #DSI.Gripper,
            DataIn := #DataIn.Gripper,
            Config := #Config.Gripper,
            Alarm := #Alarm.Gripper,
            Warning := #Warning.Gripper,
            COut => #COut.Gripper,
            DataOut => #DataOut.Gripper);
END_REGION

REGION Network 48: >
END_REGION

REGION Network 49: >
END_REGION

REGION Network 50: <<< MACHINE STATUS >>>
END_REGION

REGION Network 51: Data Out
   RUNG wire#powerrail
      I_Contact( #Ctrl.Meas1_Exe )
      I_Contact( #Ctrl.Meas2_Exe )
      Not()
      Coil( #DataOut.MeasInput_ExeReg )
   END_RUNG
   // the same network as SCL:
   #DataOut.MeasInput_ExeReg := NOT (NOT #Ctrl.Meas1_Exe AND NOT #Ctrl.Meas2_Exe);
END_REGION

REGION Network 52: Coordination Out
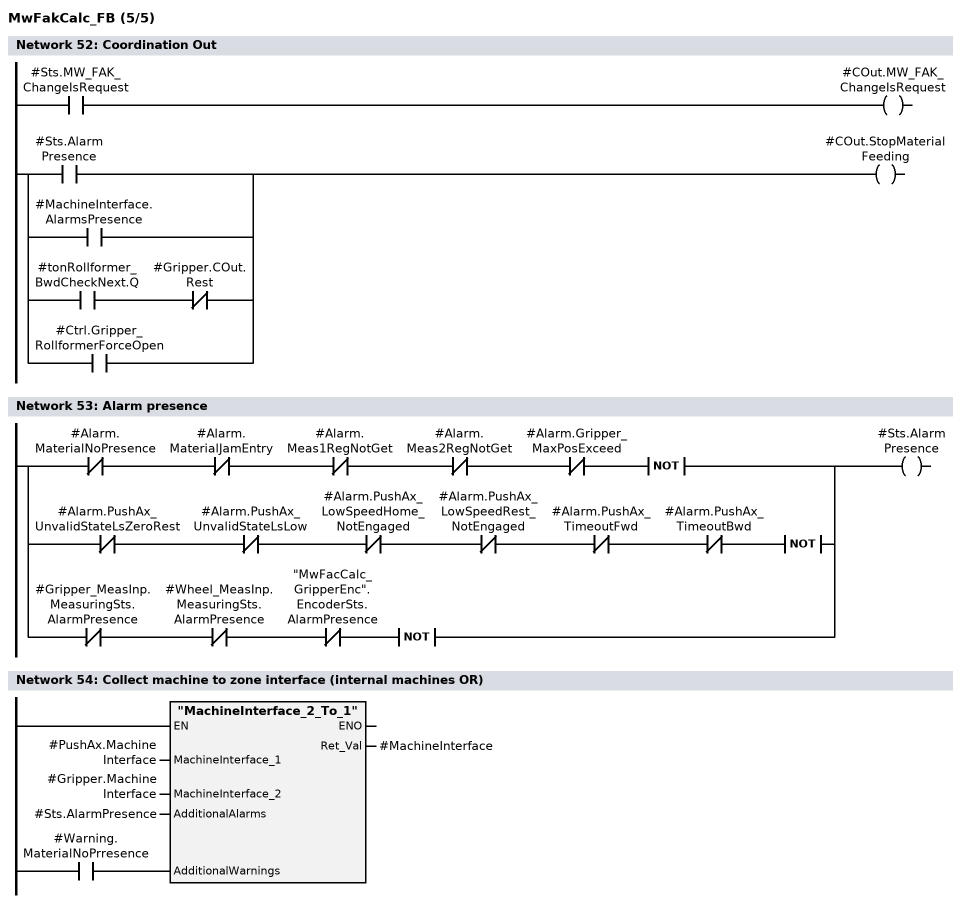
   RUNG wire#powerrail
      Contact( #Sts.MW_FAK_ChangeIsRequest )
      Coil( #COut.MW_FAK_ChangeIsRequest )
   END_RUNG
   RUNG wire#powerrail
      Contact( #Sts.AlarmPresence )
      wire#w1
      Coil( #COut.StopMaterialFeeding )
   END_RUNG
   RUNG wire#powerrail
      Contact( #MachineInterface.AlarmsPresence )
   END_RUNG wire#w1
   RUNG wire#powerrail
      Contact( #tonRollformer_BwdCheckNext.Q )
      I_Contact( #Gripper.COut.Rest )
   END_RUNG wire#w1
   RUNG wire#powerrail
      Contact( #Ctrl.Gripper_RollformerForceOpen )
   END_RUNG wire#w1
   // the same network as SCL:
   #COut.MW_FAK_ChangeIsRequest := #Sts.MW_FAK_ChangeIsRequest;
   #COut.StopMaterialFeeding := #Sts.AlarmPresence OR #MachineInterface.AlarmsPresence OR (#tonRollformer_BwdCheckNext.Q AND NOT #Gripper.COut.Rest) OR #Ctrl.Gripper_RollformerForceOpen;
END_REGION

REGION Network 53: Alarm presence
   RUNG wire#powerrail
      I_Contact( #Alarm.MaterialNoPresence )
      I_Contact( #Alarm.MaterialJamEntry )
      I_Contact( #Alarm.Meas1RegNotGet )
      I_Contact( #Alarm.Meas2RegNotGet )
      I_Contact( #Alarm.Gripper_MaxPosExceed )
      Not()
      wire#w1
      Coil( #Sts.AlarmPresence )
   END_RUNG
   RUNG wire#powerrail
      I_Contact( #Alarm.PushAx_UnvalidStateLsZeroRest )
      I_Contact( #Alarm.PushAx_UnvalidStateLsLow )
      I_Contact( #Alarm.PushAx_LowSpeedHome_NotEngaged )
      I_Contact( #Alarm.PushAx_LowSpeedRest_NotEngaged )
      I_Contact( #Alarm.PushAx_TimeoutFwd )
      I_Contact( #Alarm.PushAx_TimeoutBwd )
      Not()
   END_RUNG wire#w1
   RUNG wire#powerrail
      I_Contact( #Gripper_MeasInp.MeasuringSts.AlarmPresence )
      I_Contact( #Wheel_MeasInp.MeasuringSts.AlarmPresence )
      I_Contact( "MwFacCalc_GripperEnc".EncoderSts.AlarmPresence )
      Not()
   END_RUNG wire#w1
   // the same network as SCL:
   #Sts.AlarmPresence := NOT (NOT #Alarm.MaterialNoPresence AND NOT #Alarm.MaterialJamEntry AND NOT #Alarm.Meas1RegNotGet AND NOT #Alarm.Meas2RegNotGet AND NOT #Alarm.Gripper_MaxPosExceed) OR NOT (NOT #Alarm.PushAx_UnvalidStateLsZeroRest AND NOT #Alarm.PushAx_UnvalidStateLsLow AND NOT #Alarm.PushAx_LowSpeedHome_NotEngaged AND NOT #Alarm.PushAx_LowSpeedRest_NotEngaged AND NOT #Alarm.PushAx_TimeoutFwd AND NOT #Alarm.PushAx_TimeoutBwd) OR NOT (NOT #Gripper_MeasInp.MeasuringSts.AlarmPresence AND NOT #Wheel_MeasInp.MeasuringSts.AlarmPresence AND NOT "MwFacCalc_GripperEnc".EncoderSts.AlarmPresence);
END_REGION

REGION Network 54: Collect machine to zone interface (internal machines OR)
   RUNG wire#powerrail
      "MachineInterface_2_To_1"(AdditionalWarnings := wire#w1, MachineInterface_1 := #PushAx.MachineInterface, MachineInterface_2 := #Gripper.MachineInterface, AdditionalAlarms := #Sts.AlarmPresence, Ret_Val => #MachineInterface)
   END_RUNG
   RUNG wire#powerrail
      Contact( #Warning.MaterialNoPrresence )
   END_RUNG wire#w1
   // the same network as SCL:
   #MachineInterface := "MachineInterface_2_To_1"(MachineInterface_1 := #PushAx.MachineInterface,
                           MachineInterface_2 := #Gripper.MachineInterface,
                           AdditionalAlarms := #Sts.AlarmPresence,
                           AdditionalWarnings := #Warning.MaterialNoPrresence);
END_REGION

REGION Network 55: >
END_REGION

REGION Network 56: >
END_REGION
END_FUNCTION_BLOCK
